(* CoDeSys 2.3 export: DIR_TO_DEG.EXP *)

(* POU Engineering/conversion/DIR_TO_DEG, ST *)
FUNCTION DIR_TO_DEG : INT
VAR_INPUT
	DIR : STRING(3);
	L : INT;
END_VAR
VAR
	ly: INT;
	i : INT;
END_VAR

(*
version 1.1	22. oct. 2008
programmer 	hugo
tested by	oscat

this function converts compass directions to degrees
it will recognize up to 3 letter directions in english and german writing.

*)
IF L = 0 THEN ly := LANGUAGE.DEFAULT; ELSE ly := MIN(L, LANGUAGE.LMAX); END_IF;
FOR i := 0 TO 15 DO
	IF language.DIRS[ly, i] = DIR THEN EXIT; END_IF;
END_FOR;
DIR_TO_DEG := SHR(i * 45 + 1, 1);






(* revision histroy
hm	22. oct. 2008	rev 1.1
	original release

*)
END_FUNCTION
